% RSLogix 500 project Room_Comfort_Control_System.RSS, saved by version 8.30.00.16 %
PROJECT "UNTITLED"    % processor: Bul.1763 MicroLogix 1100 Series B %

PROGRAM FILES
  LAD 2   23 rungs

DATA FILES
  O0 OUTPUT  4 elements
  I1 INPUT  6 elements
  S2 STATUS  66 elements
  B3 BINARY  6 elements
  T4 TIMER  3 elements
  C5 COUNTER  1 elements
  R6 CONTROL  1 elements
  N7 INTEGER  2 elements
  F8 FLOAT  1 elements

LADDER 2
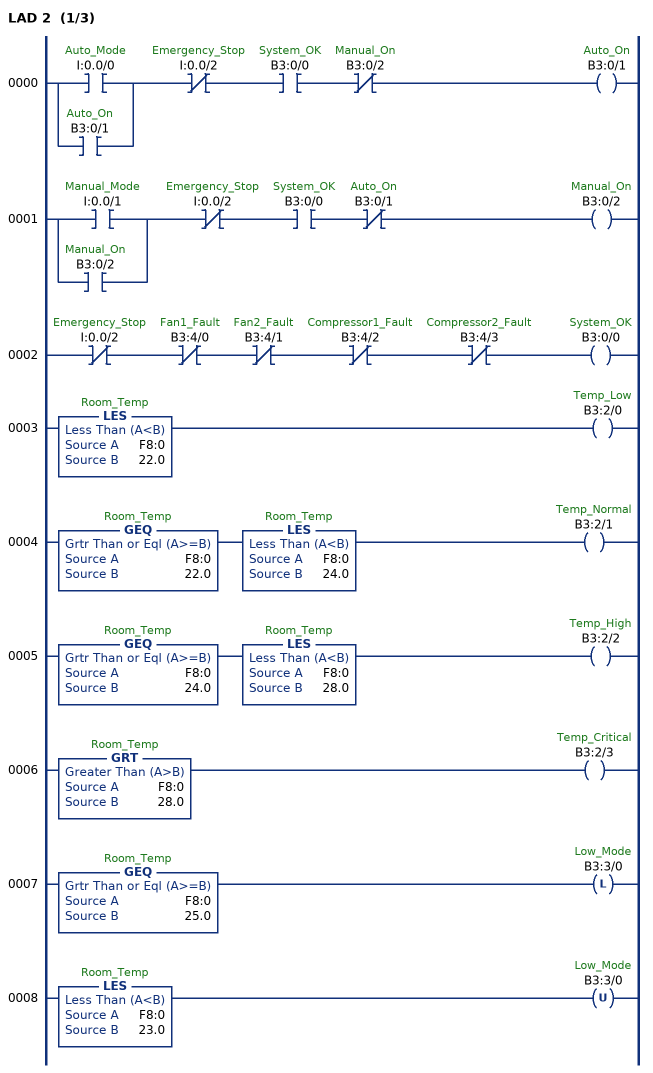
% Rung: 0 %  % edit flag set %
SOR BST XIC I:0.0/0 NXB XIC B3:0/1 BND XIO I:0.0/2 XIC B3:0/0 XIO B3:0/2 OTE B3:0/1 EOR
%   I:0.0/0  "Auto_Mode" %
%   B3:0/1  "Auto_On" %
%   I:0.0/2  "Emergency_Stop" %
%   B3:0/0  "System_OK" %
%   B3:0/2  "Manual_On" %
% Rung: 1 %  % edit flag set %
SOR BST XIC I:0.0/1 NXB XIC B3:0/2 BND XIO I:0.0/2 XIC B3:0/0 XIO B3:0/1 OTE B3:0/2 EOR
%   I:0.0/1  "Manual_Mode" %
%   B3:0/2  "Manual_On" %
%   I:0.0/2  "Emergency_Stop" %
%   B3:0/0  "System_OK" %
%   B3:0/1  "Auto_On" %
% Rung: 2 %
SOR XIO I:0.0/2 XIO B3:4/0 XIO B3:4/1 XIO B3:4/2 XIO B3:4/3 OTE B3:0/0 EOR
%   I:0.0/2  "Emergency_Stop" %
%   B3:4/0  "Fan1_Fault" %
%   B3:4/1  "Fan2_Fault" %
%   B3:4/2  "Compressor1_Fault" %
%   B3:4/3  "Compressor2_Fault" %
%   B3:0/0  "System_OK" %
% Rung: 3 %
SOR LES F8:0 22.0 OTE B3:2/0 EOR
%   F8:0  "Room_Temp" %
%   B3:2/0  "Temp_Low" %
% Rung: 4 %
SOR GEQ F8:0 22.0 LES F8:0 24.0 OTE B3:2/1 EOR
%   F8:0  "Room_Temp" %
%   B3:2/1  "Temp_Normal" %
% Rung: 5 %
SOR GEQ F8:0 24.0 LES F8:0 28.0 OTE B3:2/2 EOR
%   F8:0  "Room_Temp" %
%   B3:2/2  "Temp_High" %
% Rung: 6 %
SOR GRT F8:0 28.0 OTE B3:2/3 EOR
%   F8:0  "Room_Temp" %
%   B3:2/3  "Temp_Critical" %
% Rung: 7 %
SOR GEQ F8:0 25.0 OTL B3:3/0 EOR
%   F8:0  "Room_Temp" %
%   B3:3/0  "Low_Mode" %
% Rung: 8 %
SOR LES F8:0 23.0 OTU B3:3/0 EOR
%   F8:0  "Room_Temp" %
%   B3:3/0  "Low_Mode" %

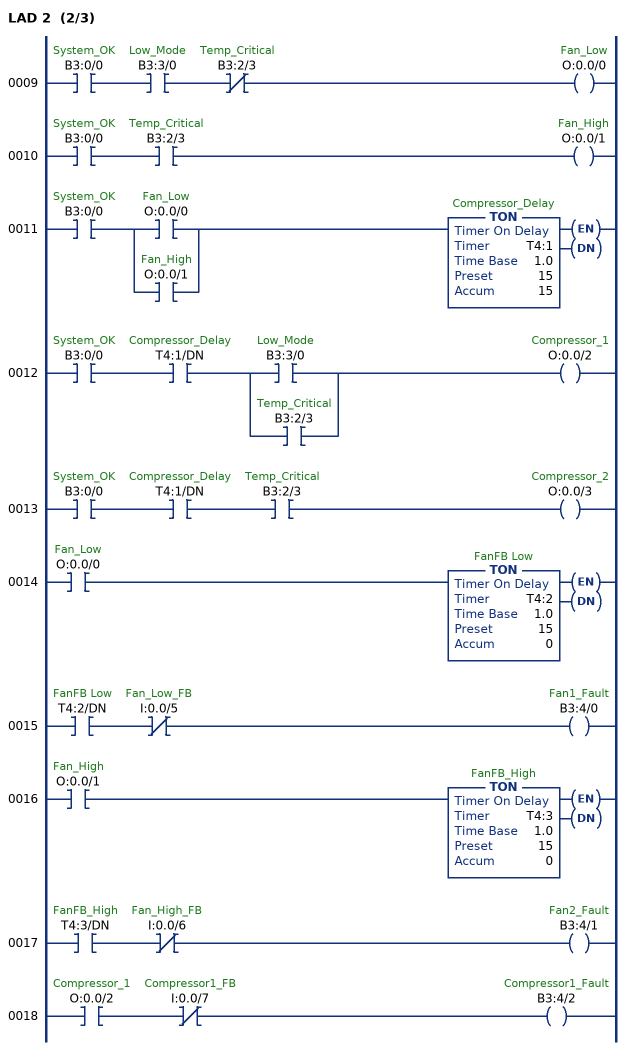
% Rung: 9 %  % edit flag set %
SOR XIC B3:0/0 XIC B3:3/0 XIO B3:2/3 OTE O:0.0/0 EOR
%   B3:0/0  "System_OK" %
%   B3:3/0  "Low_Mode" %
%   B3:2/3  "Temp_Critical" %
%   O:0.0/0  "Fan_Low" %
% Rung: 10 %  % edit flag set %
SOR XIC B3:0/0 XIC B3:2/3 OTE O:0.0/1 EOR
%   B3:0/0  "System_OK" %
%   B3:2/3  "Temp_Critical" %
%   O:0.0/1  "Fan_High" %
% Rung: 11 %  % edit flag set %
SOR XIC B3:0/0 BST XIC O:0.0/0 NXB XIC O:0.0/1 BND TON T4:1 1.0 15 15 EOR
%   B3:0/0  "System_OK" %
%   O:0.0/0  "Fan_Low" %
%   O:0.0/1  "Fan_High" %
%   T4:1  "Compressor_Delay" %
% Rung: 12 %  % edit flag set %
SOR XIC B3:0/0 XIC T4:1/DN BST XIC B3:3/0 NXB XIC B3:2/3 BND OTE O:0.0/2 EOR
%   B3:0/0  "System_OK" %
%   T4:1  "Compressor_Delay" %
%   B3:3/0  "Low_Mode" %
%   B3:2/3  "Temp_Critical" %
%   O:0.0/2  "Compressor_1" %
% Rung: 13 %  % edit flag set %
SOR XIC B3:0/0 XIC T4:1/DN XIC B3:2/3 OTE O:0.0/3 EOR
%   B3:0/0  "System_OK" %
%   T4:1  "Compressor_Delay" %
%   B3:2/3  "Temp_Critical" %
%   O:0.0/3  "Compressor_2" %
% Rung: 14 %  % edit flag set %
SOR XIC O:0.0/0 TON T4:2 1.0 15 0 EOR
%   O:0.0/0  "Fan_Low" %
%   T4:2  "FanFB Low" %
% Rung: 15 %  % edit flag set %
SOR XIC T4:2/DN XIO I:0.0/5 OTE B3:4/0 EOR
%   T4:2  "FanFB Low" %
%   I:0.0/5  "Fan_Low_FB" %
%   B3:4/0  "Fan1_Fault" %
% Rung: 16 %  % edit flag set %
SOR XIC O:0.0/1 TON T4:3 1.0 15 0 EOR
%   O:0.0/1  "Fan_High" %
%   T4:3  "FanFB_High" %
% Rung: 17 %  % edit flag set %
SOR XIC T4:3/DN XIO I:0.0/6 OTE B3:4/1 EOR
%   T4:3/DN  "FanFB_High" %
%   I:0.0/6  "Fan_High_FB" %
%   B3:4/1  "Fan2_Fault" %
% Rung: 18 %
SOR XIC O:0.0/2 XIO I:0.0/7 OTE B3:4/2 EOR
%   O:0.0/2  "Compressor_1" %
%   I:0.0/7  "Compressor1_FB" %
%   B3:4/2  "Compressor1_Fault" %

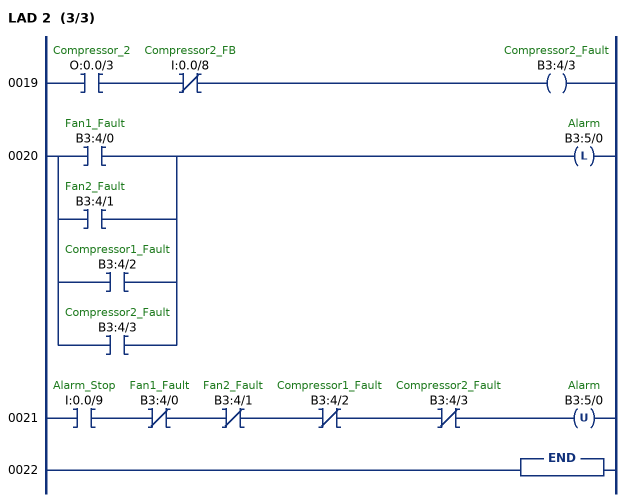
% Rung: 19 %
SOR XIC O:0.0/3 XIO I:0.0/8 OTE B3:4/3 EOR
%   O:0.0/3  "Compressor_2" %
%   I:0.0/8  "Compressor2_FB" %
%   B3:4/3  "Compressor2_Fault" %
% Rung: 20 %  % edit flag set %
SOR BST XIC B3:4/0 NXB XIC B3:4/1 NXB XIC B3:4/2 NXB XIC B3:4/3 BND OTL B3:5/0 EOR
%   B3:4/0  "Fan1_Fault" %
%   B3:4/1  "Fan2_Fault" %
%   B3:4/2  "Compressor1_Fault" %
%   B3:4/3  "Compressor2_Fault" %
%   B3:5/0  "Alarm" %
% Rung: 21 %  % edit flag set %
SOR XIC I:0.0/9 XIO B3:4/0 XIO B3:4/1 XIO B3:4/2 XIO B3:4/3 OTU B3:5/0 EOR
%   I:0.0/9  "Alarm_Stop" %
%   B3:4/0  "Fan1_Fault" %
%   B3:4/1  "Fan2_Fault" %
%   B3:4/2  "Compressor1_Fault" %
%   B3:4/3  "Compressor2_Fault" %
%   B3:5/0  "Alarm" %
% Rung: 22 %
SOR END EOR

OTHER DOCUMENTED ADDRESSES
  B3:1  "Manual_On"
  B3:1/0  "No_Emergency"
  B3:3/1  "High_Mode"
  I:1.0/0  "Auto Mode"
  I:1.0/1  "Manual Mode"
  I:2.0/2  "Emergency Stop"
  I:5.0/0  "Alarm_Stop"
  N7:0  "Room_Temp"
  N7:0/0  N  "Room_Temp"
  N7:1  "Low"
  T4:0  "Timer_1"

DATA TABLE (non-zero values as saved)
DATA B3
% B3:0 % 0X0002 0X0000 0X0004 0X0001 0X0005 0X0001
DATA T4
% .PRE .ACC %
% T4:1 % 15 15
% T4:2 % 15 0
DATA N7
% N7:0 % 24 0
